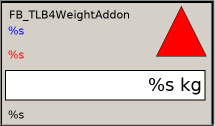
VISUALIZATION V_TLB4WeightAddon  // 215x126
VAR_IN_OUT
	{attribute 'VAR_IN_OUT_AS_POINTER'}
	fbFunction		: FB_TLB4WeightAddon;
END_VAR
    Rectangle (0,1 213x125)
    Rectangle (5,105 143x20), "%s", text variable: fbFunction.ConfigFunction.FunctionName
    Label (6,5 209x20), "FB_TLB4WeightAddon"
    Rectangle (5,21 99x20), "%s", text variable: fbFunction.WeightStates.eState
    Rectangle (5,70 200x30), "%s kg", text variable: fbFunction.Weight
    Polygon (156,56) (181,6) (206,56) (191,56) (171,56), invisible if: fbFunction.FunctionData.ErrorData.ErrorState = E_ErrorState.OPERATIONAL
    Rectangle (5,45 161x20), "%s", text variable: fbFunction.FunctionData.ErrorData.Error.ErrorCode.Conv, invisible if: fbFunction.FunctionData.ErrorData.Error.ErrorCode.Conv = 0
END_VISUALIZATION

(* stored: Version 1.1.0.1, ProductVersion 3.1.4024.4
   Visu V_TLB4WeightAddon: Id {c20c7bea-d9ff-4bc1-ae93-1b091ea39fd4} *)
